(*
Represents a component in the Entity-Component system.  
Can be cast to other interfaces for extended functionality and interaction.
*)
INTERFACE I_Component EXTENDS __SYSTEM.IQueryInterface, I_Debug

END_INTERFACE

(* stored: Version 1.1.0.1
   Itf I_Component: Id {b78f876d-df64-4417-96ac-efe56408032c} *)
